Staubli VAL3: goBeam.pgx

program goBeam()
begin
  //FUTURE ADJUSTMENT: argument nFrom
  //nFrom = 0 -> Dewar to Beam
  //nFrom = 1 -> Hotel to Beam
  movel(pHotel[0],flange,mNomSpeed)
  movel(pHotel2Beam[0],flange,mNomSpeed)
  movel(pHotel2Beam[1],flange,mNomSpeed)
  movel(pHotel2Beam[2],flange,mNomSpeed)
  movel(pHotel2Beam[3],flange,mNomSpeed)
  movel(pHotel2Beam[4],flange,mNomSpeed)
  movel(pHotel2Beam[5],flange,mNomSpeed)
  movel(pBeam,flange,mNomSpeed)
end
